Fanuc KAREL source: kt00335.KL

-- PROVISIONAL review KL for V770-1; original PC SHA256 63a989aa8e3f6ea8ef13046157642cbf31a866d41604979c376f63ad8ceb847d
-- Incomplete behavior may be omitted. Consult companion uncertainty JSON. Do not deploy.
PROGRAM KT00335
%NOLOCKGROUP
VAR
  R1 : REAL
  OUT : BOOLEAN
-- UNRESOLVED_DECL Y2 type=002018
BEGIN
  -- UNRESOLVED_PC offsets 5-16; opcodes 2E,23
  -- UNRESOLVED_PC offsets 21-35; opcodes 2E,22,9D,33,B2
  -- UNRESOLVED_PC offsets 40-63; opcodes 21,22,9D,33,B1,64,6F,23
  -- UNRESOLVED_PC offsets 68-72; opcodes 7F
END KT00335
